KUKA KRL data list: MY_SETUP.dat

&ACCESS RVP1
&REL 31
&PARAM EDITMASK = *
&PARAM TEMPLATE = C:\KRC\Roboter\Template\vorgabe
&PARAM DISKPATH = KRC:\R1\Program\_KLAVIRISTA_V2\subprogram
DEFDAT  MY_SETUP
;FOLD EXTERNAL DECLARATIONS;%{PE}%MKUKATPBASIS,%CEXT,%VCOMMON,%P
;FOLD BASISTECH EXT;%{PE}%MKUKATPBASIS,%CEXT,%VEXT,%P
EXT  BAS (BAS_COMMAND  :IN,REAL  :IN )
DECL INT counter
;ENDFOLD (BASISTECH EXT)
;FOLD USER EXT;%{E}%MKUKATPUSER,%CEXT,%VEXT,%P
;Make your modifications here

;ENDFOLD (USER EXT)
;ENDFOLD (EXTERNAL DECLARATIONS)
DECL E6POS XP1={X 212.018738,Y -176.579803,Z 442.743195,A 8.45073318,B -3.44816446,C 178.272476,S 2,T 10,E1 0.0,E2 0.0,E3 0.0,E4 0.0,E5 0.0,E6 0.0}
DECL FDAT FP1={TOOL_NO 1,BASE_NO 0,IPO_FRAME #BASE,POINT2[] " "}
DECL PDAT PPDAT1={VEL 100.000,ACC 100.000,APO_DIST 500.000,APO_MODE #CDIS,GEAR_JERK 100.000,EXAX_IGN 0}
DECL MODULEPARAM_T LAST_TP_PARAMS={PARAMS[] "Kuka.VelocityFieldEnabled=True; Kuka.ColDetectFieldEnabled=True; Kuka.MovementParameterFieldEnabled=True; Kuka.IsAngleEnabled=False; Kuka.PointName=P2; Kuka.FrameData.base_no=1; Kuka.FrameData.tool_no=4; Kuka.FrameData.ipo_frame=#BASE; Kuka.isglobalpoint=False; Kuka.MoveDataPtpName=PDAT4; Kuka.MovementDataPdat.apo_mode=#CDIS; Kuka.MovementDataPdat.apo_dist=500; Kuka.MovementData.vel=30; Kuka.MovementData.acc=100; Kuka.MovementData.exax_ign=0; Kuka.VelocityPtp=30; Kuka.BlendingEnabled=False; Kuka.APXEnabled=False; Kuka.CurrentCDSetIndex=0; Kuka.FrameData.point2=                       "}
DECL E6POS XP2={X 288.502838,Y 165.394302,Z 31.4113808,A -85.0000153,B -5.37476189E-05,C 179.900070,S 2,T 3,E1 0.0,E2 0.0,E3 0.0,E4 0.0,E5 0.0,E6 0.0}
DECL FDAT FP2={TOOL_NO 4,BASE_NO 1,IPO_FRAME #BASE,POINT2[] " "}
DECL PDAT PPDAT2={VEL 17.0000,ACC 100.000,APO_DIST 500.000,APO_MODE #CDIS,GEAR_JERK 100.000,EXAX_IGN 0}
DECL E6POS XP3={X 288.508209,Y 165.376984,Z 21.2112541,A -85.0000153,B -5.38027125E-05,C 179.900070,S 2,T 3,E1 0.0,E2 0.0,E3 0.0,E4 0.0,E5 0.0,E6 0.0}
DECL FDAT FP3={TOOL_NO 4,BASE_NO 1,IPO_FRAME #BASE,POINT2[] " "}
DECL PDAT PPDAT3={VEL 30.0000,ACC 100.000,APO_DIST 500.000,APO_MODE #CDIS,GEAR_JERK 100.000,EXAX_IGN 0}
DECL E6POS XP4={X 223.619919,Y 47.7254829,Z 442.805359,A 8.45268345,B -3.44327450,C 178.239975,S 2,T 3,E1 0.0,E2 0.0,E3 0.0,E4 0.0,E5 0.0,E6 0.0}
DECL FDAT FP4={TOOL_NO 4,BASE_NO 1,IPO_FRAME #BASE,POINT2[] " "}
DECL PDAT PPDAT4={VEL 30.0000,ACC 100.000,APO_DIST 500.000,APO_MODE #CDIS,GEAR_JERK 100.000,EXAX_IGN 0}
DECL E6POS XP5={X 136.391251,Y 151.682953,Z 50.2074394,A -85.0041122,B 0.00423473399,C 179.899353,S 2,T 2,E1 0.0,E2 0.0,E3 0.0,E4 0.0,E5 0.0,E6 0.0}
DECL FDAT FP5={TOOL_NO 4,BASE_NO 1,IPO_FRAME #BASE,POINT2[] " "}
DECL PDAT PPDAT5={VEL 50.0000,ACC 100.000,APO_DIST 500.000,APO_MODE #CDIS,GEAR_JERK 100.000,EXAX_IGN 0}
DECL E6POS XP6={X 137.135620,Y 153.937881,Z 19.7385635,A -85.0041122,B 0.00423456030,C 179.899353,S 2,T 2,E1 0.0,E2 0.0,E3 0.0,E4 0.0,E5 0.0,E6 0.0}
DECL FDAT FP6={TOOL_NO 4,BASE_NO 1,IPO_FRAME #BASE,POINT2[] " "}
DECL PDAT PPDAT6={VEL 30.0000,ACC 100.000,APO_DIST 500.000,APO_MODE #CDIS,GEAR_JERK 100.000,EXAX_IGN 0}
DECL E6POS XP7={X 137.133301,Y 153.945404,Z 24.1670036,A -85.0041122,B 0.00426238682,C 179.899063,S 2,T 2,E1 0.0,E2 0.0,E3 0.0,E4 0.0,E5 0.0,E6 0.0}
DECL FDAT FP7={TOOL_NO 4,BASE_NO 1,IPO_FRAME #BASE,POINT2[] " "}
DECL PDAT PPDAT7={VEL 30.0000,ACC 100.000,APO_DIST 500.000,APO_MODE #CDIS,GEAR_JERK 100.000,EXAX_IGN 0}
DECL PDAT PPDAT9={VEL 30.0000,ACC 100.000,APO_DIST 500.000,APO_MODE #CDIS,GEAR_JERK 100.000,EXAX_IGN 0}
DECL FDAT FP9={TOOL_NO 1,BASE_NO 0,IPO_FRAME #BASE,POINT2[] " "}
DECL E6POS XP9={X 238.631805,Y -103.017105,Z 431.766388,A 8.45245838,B -3.44352770,C 178.244766,S 2,T 10,E1 0.0,E2 0.0,E3 0.0,E4 0.0,E5 0.0,E6 0.0}
DECL PDAT PPDAT8={VEL 30.0000,ACC 100.000,APO_DIST 500.000,APO_MODE #CDIS,GEAR_JERK 100.000,EXAX_IGN 0}
DECL FDAT FP8={TOOL_NO 1,BASE_NO 0,IPO_FRAME #BASE,POINT2[] " "}
DECL E6POS XP8={X 239.692657,Y -103.017105,Z 425.322327,A 8.45245838,B -3.44352770,C 178.244766,S 2,T 10,E1 0.0,E2 0.0,E3 0.0,E4 0.0,E5 0.0,E6 0.0}
ENDDAT
